/// User-facing logging interface.
/// Implemented by `DefaultLogger` and any test doubles.
///
/// For structured attributes use the concrete `DefaultLogger` type directly,
/// which adds `WithAttribute` and `OnCondition` chaining methods.
INTERFACE PUBLIC Logger EXTENDS __System.IQueryInterface

/// Log at DEBUG level.
METHOD PUBLIC Debug : BOOL
VAR_INPUT
	message : Tc2_System.T_MaxString;
END_VAR
END_METHOD

/// Log at ERROR level.
METHOD PUBLIC Error : BOOL
VAR_INPUT
	message : Tc2_System.T_MaxString;
END_VAR
END_METHOD

/// Log at FATAL level.
METHOD PUBLIC Fatal : BOOL
VAR_INPUT
	message : Tc2_System.T_MaxString;
END_VAR
END_METHOD

/// Log at INFORMATION level.
METHOD PUBLIC Info : BOOL
VAR_INPUT
	message : Tc2_System.T_MaxString;
END_VAR
END_METHOD

/// Log at WARNING level.
METHOD PUBLIC Warning : BOOL
VAR_INPUT
	message : Tc2_System.T_MaxString;
END_VAR
END_METHOD

END_INTERFACE

(* stored: Version 1.1.0.1
   Itf Logger: Id {142e5ac4-9651-4b60-842f-9fed1e0c8704}
   Method Debug: Id {f6a7b8c9-d0e1-2345-f012-456789012345}
   Method Error: Id {c9d0e1f2-a3b4-5678-2345-789012345678}
   Method Fatal: Id {d0e1f2a3-b4c5-6789-3456-890123456789}
   Method Info: Id {a7b8c9d0-e1f2-3456-0123-567890123456}
   Method Warning: Id {b8c9d0e1-f2a3-4567-1234-678901234567} *)
